{attribute 'qualified_only'}
{attribute 'strict'}
{attribute 'to_string'}
TYPE E_CompositeServiceErrorCode :
(
	None := 0,
	NotConfigured := 1,
	OwnershipConflict := 2,
	DependencyNotIdle := 3,
	UnsupportedCompletionBehavior := 4,
	InternalCallSubmitFailed := 5,
	InternalCommandRejected := 6,
	ChildStoppedUnexpectedly := 7,
	ChildAbortedUnexpectedly := 8,
	SequenceFailed := 9,
	InvalidSequenceState := 10
) UDINT;
END_TYPE

(* stored: Version 1.1.0.1, ProductVersion 3.1.4026.18
   DUT E_CompositeServiceErrorCode: Id {60869512-0163-482e-8555-0c0b975e1b79} *)
